FUNCTION_BLOCK Motor_Sorting
VAR_INPUT
	Inp_Conveyor_2_Palette_Right_Side_at_Sorter						: BOOL;	
	Inp_Sortierer_in_Basic_Position									: BOOL;
	Inp_Sorter_Plunger_Above										: BOOL;
	Inp_Sorter_Plunger_Below										: BOOL;
	Inp_Measuring_Bar_Sorting_Axis_X								: INT;
	Inp_Measuring_Bar_Sorting_Axis_Y								: INT;
	Inp_Form_is_Changed_Button										: BOOL;
END_VAR
VAR_OUTPUT
	Out_Sorter_Pluger_Drive_Up										: BOOL;	
	Out_Sorter_Pluger_Drive_Down									: BOOL;	
	Out_Measuring_Bar_Sorting_Axis_X_Right_Rotation_Motor_On		: BOOL;
	Out_Measuring_Bar_Sorting_Axis_Y_Right_Rotation_Motor_On		: BOOL;
	Out_Measuring_Bar_Sorting_Axis_X_Left_Rotation_Motor_On			: BOOL;
	Out_Measuring_Bar_Sorting_Axis_Y_Left_Rotation_Motor_On			: BOOL;
	Out_Sorter_Pluger_Pull_in										: BOOL;	
	Palette_at_Sorter_is_free										: BOOL;
END_VAR
VAR
	positions_init													: Positions_init;
	Pluger_Below_TON_For_Drive										: TON;
	Pluger_Below_TON_For_Release									: TON;
	i																: INT := 1;
	Measuring_Bar_Sorting_Axis_X_Motor_Above_Sorting_Place			: BOOL;
	Measuring_Bar_Sorting_Axis_Y_Motor_Above_Sorting_Place			: BOOL;
	Measuring_Bar_Sorting_Axis_X_Motor_At_Start_Position			: BOOL;
	Measuring_Bar_Sorting_Axis_Y_Motor_At_Start_Position			: BOOL;
	Part_On_Place													: BOOL;
	Part_on_Palette_at_Sorter										: BOOL;
	Part_Is_taken													: BOOL;
	Form_for_parts_is_FULL: BOOL;
END_VAR

positions_init();
Pluger_Below_TON_For_Drive(IN:= The_Sorter_is_ready_for_sorting() AND Inp_Sorter_Plunger_Below, PT:= T#2S);
Pluger_Below_TON_For_Release(IN:= Measuring_Bar_Sorting_Axis_X_Motor_Above_Sorting_Place 
	AND Measuring_Bar_Sorting_Axis_Y_Motor_Above_Sorting_Place AND Part_On_Place AND Inp_Sorter_Plunger_Below, PT:= T#2S);

//If Form is full
IF i<=9 THEN Form_for_parts_is_FULL:=TRUE;i:=0;	
END_IF

IF Inp_Form_is_Changed_Button AND i<9
	THEN Form_for_parts_is_FULL:=FALSE;
END_IF

//Step 1 : Plunger goes down for a Part
IF The_Sorter_is_ready_for_sorting() AND Main.conveyor_2.M_Part_is_ready_for_sorting 
AND Inp_Sorter_Plunger_Above AND Part_on_Palette_at_Sorter AND NOT Form_for_parts_is_FULL 
	THEN Out_Sorter_Pluger_Drive_Up:=FALSE; 
	Out_Sorter_Pluger_Drive_Down:=TRUE;
	Part_On_Place:=FALSE;
END_IF

//Step 2 : Plunger takes a Part
IF The_Sorter_is_ready_for_sorting() AND Inp_Sorter_Plunger_Below
	THEN Out_Sorter_Pluger_Pull_in:=TRUE; Part_on_Palette_at_Sorter:=FALSE;
END_IF

//Step 3 : Plunger is waiting for a 2 Seconds and drives up
IF The_Sorter_is_ready_for_sorting() AND Pluger_Below_TON_For_Drive.Q
	THEN 
	Out_Sorter_Pluger_Drive_Down:=FALSE;
	Out_Sorter_Pluger_Drive_Up:=TRUE;
	Part_Is_taken:=TRUE;
END_IF

//Step 4 : Plunger goes to Parts place
IF The_Sorter_is_ready_for_sorting() AND Inp_Sorter_Plunger_Above AND Part_Is_taken
	THEN to_Parts_Place(); Palette_at_Sorter_is_free:=TRUE;
END_IF

//Step 5 : Plunger puts Part to place
IF Measuring_Bar_Sorting_Axis_X_Motor_Above_Sorting_Place 
	AND Measuring_Bar_Sorting_Axis_Y_Motor_Above_Sorting_Place
	AND Inp_Sorter_Plunger_Above
	THEN 
	Out_Sorter_Pluger_Drive_Up:=FALSE;
	Out_Sorter_Pluger_Drive_Down:=TRUE;	
END_IF

//Step 6 : Plunger releases Part
IF Measuring_Bar_Sorting_Axis_X_Motor_Above_Sorting_Place 
	AND Measuring_Bar_Sorting_Axis_Y_Motor_Above_Sorting_Place AND Inp_Sorter_Plunger_Below
	THEN 
	Out_Sorter_Pluger_Pull_in:=FALSE;
	Part_On_Place:=TRUE;
END_IF

//Step 7 : Plunger releases Part
IF Pluger_Below_TON_For_Release.Q
	THEN 
	Out_Sorter_Pluger_Drive_Down:=FALSE;
	Out_Sorter_Pluger_Drive_Up:=TRUE;
	Part_Is_taken:=FALSE;
END_IF

//Step 7 : Sorter goes to the start position
IF Measuring_Bar_Sorting_Axis_X_Motor_Above_Sorting_Place 
	AND Measuring_Bar_Sorting_Axis_Y_Motor_Above_Sorting_Place
	AND Inp_Sorter_Plunger_Above
 	AND Part_On_Place 
	AND Part_Is_taken=FALSE
	THEN 
	to_Start();
	GVL.Part_is_Sorted:=TRUE;
END_IF

METHOD PRIVATE The_Sorter_is_ready_for_sorting : BOOL
VAR_INPUT
END_VAR
IF 	Measuring_Bar_Sorting_Axis_X_Motor_At_Start_Position AND
	Measuring_Bar_Sorting_Axis_Y_Motor_At_Start_Position
AND Inp_Conveyor_2_Palette_Right_Side_at_Sorter
THEN The_Sorter_is_ready_for_sorting:=TRUE;
END_IF

IF 	Measuring_Bar_Sorting_Axis_X_Motor_At_Start_Position =FALSE OR
	Measuring_Bar_Sorting_Axis_Y_Motor_At_Start_Position =FALSE
OR Inp_Conveyor_2_Palette_Right_Side_at_Sorter  =FALSE
THEN The_Sorter_is_ready_for_sorting:=FALSE;
END_IF
END_METHOD

ACTION to_Parts_Place:
FOR i :=1 TO 9 DO
	IF Inp_Measuring_Bar_Sorting_Axis_X < positions_init.Current_Position[i].Coordinate_X_Axis
		THEN Out_Measuring_Bar_Sorting_Axis_X_Right_Rotation_Motor_On:=TRUE;
Measuring_Bar_Sorting_Axis_X_Motor_Above_Sorting_Place:=FALSE; 
	END_IF
	IF Inp_Measuring_Bar_Sorting_Axis_X >= positions_init.Current_Position[i].Coordinate_X_Axis
		THEN Out_Measuring_Bar_Sorting_Axis_X_Right_Rotation_Motor_On:=FALSE; 
			Measuring_Bar_Sorting_Axis_X_Motor_Above_Sorting_Place:=TRUE;
	END_IF
	
		IF Inp_Measuring_Bar_Sorting_Axis_Y < positions_init.Current_Position[i].Coordinate_Y_Axis
		THEN Out_Measuring_Bar_Sorting_Axis_Y_Right_Rotation_Motor_On:=TRUE;
		Measuring_Bar_Sorting_Axis_X_Motor_Above_Sorting_Place:=FALSE; 
	END_IF
	IF Inp_Measuring_Bar_Sorting_Axis_Y >= positions_init.Current_Position[i].Coordinate_Y_Axis
		THEN Out_Measuring_Bar_Sorting_Axis_Y_Right_Rotation_Motor_On:=FALSE; 
			Measuring_Bar_Sorting_Axis_Y_Motor_Above_Sorting_Place:=TRUE;
	END_IF
END_FOR
END_ACTION

ACTION to_Start:
	IF Inp_Measuring_Bar_Sorting_Axis_X > positions_init.Current_Position[0].Coordinate_X_Axis
		THEN Out_Measuring_Bar_Sorting_Axis_X_Left_Rotation_Motor_On:=TRUE; 
	END_IF
	IF Inp_Measuring_Bar_Sorting_Axis_X <= positions_init.Current_Position[0].Coordinate_X_Axis
		THEN Out_Measuring_Bar_Sorting_Axis_X_Left_Rotation_Motor_On:=FALSE; 
			Measuring_Bar_Sorting_Axis_X_Motor_At_Start_Position:=TRUE;
	END_IF
	
		IF Inp_Measuring_Bar_Sorting_Axis_Y > positions_init.Current_Position[0].Coordinate_Y_Axis
		THEN Out_Measuring_Bar_Sorting_Axis_Y_Left_Rotation_Motor_On:=TRUE;
	END_IF
	IF Inp_Measuring_Bar_Sorting_Axis_Y <= positions_init.Current_Position[0].Coordinate_Y_Axis
		THEN Out_Measuring_Bar_Sorting_Axis_Y_Left_Rotation_Motor_On:=FALSE; 
			Measuring_Bar_Sorting_Axis_Y_Motor_At_Start_Position:=TRUE;
	END_IF
END_ACTION

END_FUNCTION_BLOCK

(* stored: Version 1.1.0.1, ProductVersion 3.1.4024.12
   POU Motor_Sorting: Id {bf82215d-3dde-493f-ab69-71f13ec01e05}, SpecialFunc None
   Method The_Sorter_is_ready_for_sorting: Id {6482a0e9-f631-4496-a3c5-89d8235978d6}
   Action to_Parts_Place: Id {c17ccfb0-8731-4c60-b1c6-1c1220e803bc}
   Action to_Start: Id {898dc70e-a19e-452a-b1ae-fdbf47edb521} *)
